// TwinCAT 3 PLC project tcext
// Title: TcExt
// Company: TcExt
// ProjectVersion: 0.2.3
// ProgramVersion: 3.1.4022.7
// libraries:
//   Tc2_Standard, * (Beckhoff Automation GmbH)
//   Tc2_System, * (Beckhoff Automation GmbH)
//   Tc2_Utilities, * (Beckhoff Automation GmbH)
//   Tc3_Module, * (Beckhoff Automation GmbH)
//   TcUnit, * (www.tcunit.org)
// project tree:
//   Files/ FileMemory.TcPOU, FileMemoryAction.TcDUT
//   Object/ BitAdrState.TcPOU, ModabsInt.TcPOU, Object.TcPOU
//   Tests/Files/ TestFileMemory.TcPOU
//   Tests/ MAIN.TcPOU, MAIN_TEST.TcPOU, PlcTask.TcTTO, TestBitAdrState.TcPOU, TestModabsInt.TcPOU
//   Tests/Timer/ TestSignalDutyCycleRecorder.TcPOU
//   Timer/ GetSystemTimeAsTime.TcPOU, SignalTimeRecorder.TcPOU, SignalDutyCycleRecorder.TcPOU, SimpleSignalTimeRecorder.TcPOU, SimpleTimeRecorder.TcPOU
//   Utils/ CompareReal.TcPOU, CrcCheck.TcPOU, FlashSignal.TcPOU, LockingRelay.TcPOU, TransitionController.TcPOU
//   Visu/ Colors.TcDUT, VisuElementProperties.TcDUT
// real-time tasks:
//   TASK PlcTask: cycle T#10ms, priority 20, ADS port 351

CONFIGURATION tcext
    RESOURCE PLC ON TwinCAT3
        TASK PlcTask(INTERVAL := T#10ms, PRIORITY := 20);
        PROGRAM MAIN WITH PlcTask : MAIN;
    END_RESOURCE
END_CONFIGURATION

// ---- Files/FileMemoryAction.TcDUT
{attribute 'qualified_only'}
{attribute 'strict'}
TYPE FileMemoryAction :
(
	UNLOCKED := 0,
  READ,
  WRITE
);
END_TYPE

// ---- Visu/Colors.TcDUT
{attribute 'qualified_only'}
{attribute 'strict'}
TYPE Colors :
(
  WHITE := 16#FFFFFF,
	BLACK := 16#000000,
	GRAY := 16#4C4C4C,
	LIGHT_GRAY := 16#C0C0C0,
	DARK_GRAY := 16#2D2D2D,
	RED := 16#FF0000,
	GREEN := 16#00FF00,
	YELLOW := 16#FFFF00,
  BLUE := 16#00BFFF
) DWORD := WHITE;
END_TYPE

// ---- Visu/VisuElementProperties.TcDUT
TYPE VisuElementProperties :
STRUCT
  color: DWORD;
  invisible: BOOL;
  int_value: INT;
END_STRUCT
END_TYPE

// ---- Tests/MAIN.TcPOU
{attribute 'hide'}
PROGRAM MAIN
VAR
END_VAR

{IF defined(TEST)}
MAIN_TEST();
{END_IF}

END_PROGRAM

// ---- Tests/MAIN_TEST.TcPOU
{attribute 'hide'}
PROGRAM MAIN_TEST
VAR
  test_file_memory: TestFileMemory;
  test_durchflusssensor: TestSignalDutyCycleRecorder;
  time_test: TIME;
  test_bit_adr_state: TestBitAdrState;
  test_modabs_int: TestModabsInt;
END_VAR

TcUnit.RUN();
time_test := TO_TIME(F_GetSystemTime()/10000);

END_PROGRAM

// ---- Tests/Files/TestFileMemory.TcPOU
{attribute 'call_after_init'}
FUNCTION_BLOCK TestFileMemory EXTENDS TcUnit.FB_TestSuite
VAR
END_VAR

//createFile();
set_path();
write_file();
read_non_existent_file();
read_existent_file();
write_and_read_simultaneously();
read_twice();
write_twice();
auto_write();
auto_write_time();

METHOD auto_write
VAR
  done: BOOL;
  error_id: UDINT;
END_VAR
VAR_INST
  file_memory: FileMemory;
  test_data: INT;
  test_data_first_read: INT;
  test_data_second_read: INT;
  counter: INT;
END_VAR
TEST('auto_write');

file_memory.path := 'c:\auto_write.be';
file_memory.auto_write(
  data_ptr:=ADR(test_data),
  data_size:=SIZEOF(test_data),
  done=>done,
  error_id=>error_id);

CASE counter OF
0:
  test_data := 135;
  counter := counter + 10;
10:
  IF done THEN
    counter := counter + 10;
  END_IF
20:
  file_memory.read(
    start:=TRUE,
    data_ptr:=ADR(test_data_first_read),
    data_size:=SIZEOF(test_data_first_read),
    done=>done,
    error_id=>error_id);
  IF done THEN
    counter := counter + 10;
  END_IF
30:
  file_memory.read(
    start:=FALSE,
    data_ptr:=0,
    data_size:=0);
  counter := counter + 10;
40:
  test_data := 246;
  counter := counter + 10;
50:
  IF done THEN
    counter := counter + 10;
  END_IF
60:
  file_memory.read(
    start:=TRUE,
    data_ptr:=ADR(test_data_second_read),
    data_size:=SIZEOF(test_data_second_read),
    done=>done,
    error_id=>error_id);
  IF done THEN
    AssertEquals_INT(135, test_data_first_read, 'Wrong values from auto_write file.');
    AssertEquals_INT(246, test_data_second_read, 'Wrong values from auto_write file.');
  
    TEST_FINISHED();
  END_IF
END_CASE
END_METHOD

METHOD auto_write_time
VAR
  done: BOOL;
  error_id: UDINT;
END_VAR
VAR_INST
  file_memory: FileMemory;
  test_data: INT;
  test_data_first_read: INT;
  test_data_second_read: INT;
  counter: INT;
  test_timer: TON;
END_VAR
TEST('auto_write_time');

file_memory.path := 'c:\auto_write_time.be';
file_memory.auto_write_time(
  data_ptr:=ADR(test_data),
  data_size:=SIZEOF(test_data),
  period:=T#2S,
  done=>done,
  error_id=>error_id);
test_timer(PT:=T#2.2S);

CASE counter OF
0:
  test_data := 135;
  counter := counter + 10;
10:
  test_timer(IN:=TRUE);
  IF test_timer.q THEN
    test_timer(IN:=FALSE);
    counter := counter + 10;
  END_IF
20:
  file_memory.read(
    start:=TRUE,
    data_ptr:=ADR(test_data_first_read),
    data_size:=SIZEOF(test_data_first_read),
    done=>done,
    error_id=>error_id);
  IF done THEN
    counter := counter + 10;
  END_IF
30:
  file_memory.read(
    start:=FALSE,
    data_ptr:=0,
    data_size:=0);
  counter := counter + 10;
40:
  test_data := 246;
  counter := counter + 10;
50:
  test_timer(IN:=TRUE);
  IF test_timer.q THEN
    test_timer(IN:=FALSE);
    counter := counter + 10;
  END_IF
60:
  file_memory.read(
    start:=TRUE,
    data_ptr:=ADR(test_data_second_read),
    data_size:=SIZEOF(test_data_second_read),
    done=>done,
    error_id=>error_id);
  IF done THEN
    AssertEquals_INT(135, test_data_first_read, 'Wrong values from auto_write file.');
    AssertEquals_INT(246, test_data_second_read, 'Wrong values from auto_write file.');
  
    TEST_FINISHED();
  END_IF
END_CASE
END_METHOD

METHOD PRIVATE createFile
VAR_INPUT
END_VAR
TEST('create_file');

TEST_FINISHED();
END_METHOD

METHOD read_existent_file
VAR
  done: BOOL;
  error_id: UDINT;
  
  expected: INT;
END_VAR
VAR_INST
  file_memory: FileMemory;
  test_data: INT;
END_VAR
TEST('read_existent_file');

IF IS_TEST_FINISHED('write_file') THEN
  file_memory.path := 'c:\test_file.be';
  
  file_memory.read(
    start:=TRUE,
    data_ptr:=ADR(test_data),
    data_size:=SIZEOF(test_data),
    done=>done,
    error_id=>error_id);
  
  IF done THEN
    expected := 37;
    AssertEquals_INT(expected, test_data, CONCAT('Wrong value. Check if file exists and contains 37. Error: ', TO_STRING(error_id)));
    
    TEST_FINISHED();
  END_IF
END_IF
END_METHOD

METHOD PRIVATE read_non_existent_file
VAR
  done: BOOL;
  error_id: UDINT;
  
  test_data: INT;
END_VAR
VAR_INST
    read_file: FileMemory;
END_VAR
TEST('read_non_existent_file');

read_file.path := 'c:\non_existent_file.be';

read_file.read(
  start:=TRUE,
  data_ptr:=ADR(test_data),
  data_size:=SIZEOF(test_data),
  done=>done,
  error_id=>error_id);

IF done THEN
  AssertTrue((error_id <> 0), 'No error although file non existent.');
  
  TEST_FINISHED();
END_IF
END_METHOD

METHOD read_twice
VAR
  done: BOOL;
  error_id: UDINT;
END_VAR
VAR_INST
  file_memory: FileMemory;
  test_data_first_read: INT;
  test_data_second_read: INT;
  counter: INT;
END_VAR
TEST('read_twice');

IF IS_TEST_FINISHED('write_file') AND IS_TEST_FINISHED('read_existent_file') THEN
  file_memory.path := 'c:\test_file.be';
  
  CASE counter OF
  0:
    file_memory.read(
      start:=TRUE,
      data_ptr:=ADR(test_data_first_read),
      data_size:=SIZEOF(test_data_first_read),
      done=>done,
      error_id=>error_id);
    IF done THEN
      counter := 10;
		END_IF
  10:
    file_memory.read(
      start:=FALSE,
      data_ptr:=0,
      data_size:=0);
    counter := 20;
  20:
    file_memory.read(
      start:=TRUE,
      data_ptr:=ADR(test_data_second_read),
      data_size:=SIZEOF(test_data_second_read),
      done=>done,
      error_id=>error_id);
    IF done THEN
      AssertEquals_INT(test_data_first_read, test_data_second_read, 'Wrong values from same file.');
    
      TEST_FINISHED();
		END_IF
	END_CASE
END_IF
END_METHOD

METHOD set_path
VAR
  actual: STRING;
  expected: STRING;
  
  file_memory: FileMemory;
END_VAR
TEST('set_path');

expected := 'c:\test.be';
file_memory.path := expected;
actual := file_memory.path;

AssertEquals_STRING(expected, actual, 'Path is broken.');

TEST_FINISHED();
END_METHOD

METHOD write_and_read_simultaneously
VAR
  done_write: BOOL;
  error_id_write: UDINT;
  done_read: BOOL;
  error_id_read: UDINT;
END_VAR
VAR_INST
  file_memory: FileMemory;
  test_data_write: INT;
  test_data_read: INT;
END_VAR
TEST('write_and_read_simultaneously');

file_memory.path := 'c:\test_file_2.be';

test_data_write := 123;
file_memory.write(
  start:=TRUE , 
  data_ptr:=ADR(test_data_write), 
  data_size:=SIZEOF(test_data_write), 
  done=>done_write, 
  error_id=>error_id_write);
file_memory.read(
  start:=TRUE , 
  data_ptr:=ADR(test_data_read), 
  data_size:=SIZEOF(test_data_read), 
  done=>done_read, 
  error_id=>error_id_read);
  
IF done_write AND done_read THEN
  AssertTrue((error_id_write = 0), CONCAT('Fehler beim simultanen Schreiben. Error: ', TO_STRING(error_id_write)));
  AssertTrue((error_id_read = 0), CONCAT('Fehler beim simultanen Lesen. Error: ', TO_STRING(error_id_read)));
  AssertEquals_INT(test_data_write, test_data_read, 'Geschriebene und gelesenen Daten ungleich.');
  
  TEST_FINISHED();
END_IF
END_METHOD

METHOD write_file
VAR
  done: BOOL;
  error_id: UDINT;
END_VAR
VAR_INST
  file_memory: FileMemory;
  test_data: INT;
END_VAR
TEST('write_file');

file_memory.path := 'c:\test_file.be';

test_data := 37;

file_memory.write(
  start:=TRUE,
  data_ptr:=ADR(test_data),
  data_size:=SIZEOF(test_data),
  done=>done,
  error_id=>error_id);
  
IF done THEN
  AssertEquals_UDINT(0, error_id, CONCAT('File could not be written. Error: ', TO_STRING(error_id)));
  
  TEST_FINISHED();
END_IF
END_METHOD

METHOD write_twice
VAR
  done: BOOL;
  error_id: UDINT;
END_VAR
VAR_INST
  file_memory: FileMemory;
  test_data_first_write: INT;
  test_data_second_write: INT;
  test_data_first_read: INT;
  test_data_second_read: INT;
  counter: INT;
END_VAR
TEST('write_twice');

file_memory.path := 'c:\write_twice.be';

test_data_first_write := 123;
test_data_second_write := 456;
CASE counter OF
0:
  file_memory.write(
    start:=TRUE,
    data_ptr:=ADR(test_data_first_write),
    data_size:=SIZEOF(test_data_first_write),
    done=>done,
    error_id=>error_id);
  IF done THEN
    counter := 10;
  END_IF
10:
  file_memory.write(
    start:=FALSE,
    data_ptr:=0,
    data_size:=0);
  counter := 20;
20:
  file_memory.read(
    start:=TRUE,
    data_ptr:=ADR(test_data_first_read),
    data_size:=SIZEOF(test_data_first_read),
    done=>done,
    error_id=>error_id);
  IF done THEN
    counter := 30;
  END_IF
30:
  file_memory.read(
    start:=FALSE,
    data_ptr:=0,
    data_size:=0);
  counter := 40;
40:
  file_memory.write(
    start:=TRUE,
    data_ptr:=ADR(test_data_second_write),
    data_size:=SIZEOF(test_data_second_write),
    done=>done,
    error_id=>error_id);
  IF done THEN
    counter := 50;
  END_IF
50:
  file_memory.write(
    start:=FALSE,
    data_ptr:=0,
    data_size:=0);
  counter := 60;
60:
  file_memory.read(
    start:=TRUE,
    data_ptr:=ADR(test_data_second_read),
    data_size:=SIZEOF(test_data_second_read),
    done=>done,
    error_id=>error_id);
  IF done THEN
    AssertEquals_INT(test_data_first_write, test_data_first_read, 'Wrong values from same file.');
    AssertEquals_INT(test_data_second_write, test_data_second_read, 'Wrong values from same file.');
  
    TEST_FINISHED();
  END_IF
END_CASE
END_METHOD

END_FUNCTION_BLOCK

// ---- Files/FileMemory.TcPOU
FUNCTION_BLOCK FileMemory EXTENDS Object
VAR
  file_path: Tc2_System.T_MaxString;
  
  fb_file_open: Tc2_System.FB_FileOpen;
  fb_file_close: Tc2_System.FB_FileClose;
  fb_file_read: Tc2_System.FB_FileRead;
  fb_file_write: Tc2_System.FB_FileWrite;
  
  t_timeout_read: TIME := T#2S;
  t_timeout_write: TIME := T#2S;
  
  lock_action: FileMemoryAction;
  
  write_period_timer: Tc2_Standard.TP;
  crc_check: CrcCheck;
  _mode_read: DWORD := Tc2_System.FOPEN_MODEREAD OR Tc2_System.FOPEN_MODEBINARY;
  _mode_write: DWORD := Tc2_System.FOPEN_MODEWRITE OR Tc2_System.FOPEN_MODEBINARY;
END_VAR

METHOD auto_write
VAR_INPUT
  data_ptr: POINTER TO BYTE;
  data_size: UDINT;
END_VAR
VAR_OUTPUT
  done: BOOL;
  error_id: UDINT;
END_VAR
VAR
  crc_changed: BOOL;
END_VAR
VAR_INST
  act_crc: UINT;
  previous_crc: UINT;
END_VAR
write(
  start:=crc_check.data_changed(data_ptr, data_size), 
  data_ptr:=data_ptr, 
  data_size:=data_size,
  done=>done,
  error_id=>error_id);
  
IF done THEN
  crc_check.reset();
END_IF
END_METHOD

METHOD auto_write_time
VAR_INPUT
  data_ptr: POINTER TO BYTE;
  data_size: UDINT;
  period: TIME;
END_VAR
VAR_OUTPUT
  done: BOOL;
  error_id: UDINT;
END_VAR
write_period_timer(IN:=NOT write_period_timer.Q, PT:=period);

write(
  start:=NOT write_period_timer.q AND crc_check.data_changed(data_ptr, data_size), 
  data_ptr:=data_ptr, 
  data_size:=data_size,
  done=>done,
  error_id=>error_id);
  
IF NOT write_period_timer.q THEN
  crc_check.reset();
END_IF
END_METHOD

PROPERTY PUBLIC busy_reading : BOOL
GET
busy_reading := THIS^.lock_action = FileMemoryAction.READ;
END_GET
END_PROPERTY

PROPERTY PUBLIC busy_writing : BOOL
GET
busy_writing := THIS^.lock_action = FileMemoryAction.WRITE;
END_GET
END_PROPERTY

METHOD file_close
VAR_INPUT
  start: BOOL;
  file_handler: UINT;
END_VAR
VAR_OUTPUT
  done: BOOL;
  error_id: UDINT;
END_VAR
fb_file_close(
  bExecute:=start,
  hFile:=file_handler);

IF NOT fb_file_close.bBusy THEN
  done := TRUE;
  IF fb_file_close.bError THEN
    error_id := fb_file_close.nErrId;
  END_IF
END_IF
END_METHOD

METHOD PRIVATE file_open: UINT
VAR_INPUT
  start: BOOL;
  mode: DWORD;
END_VAR
VAR_OUTPUT
  done: BOOL;
  error_id: UDINT;
END_VAR
fb_file_open(
  bExecute:=start,
  sPathName:=path,
  nMode:=mode);

file_open := 0;
IF NOT fb_file_open.bBusy THEN
  done := TRUE;
  IF fb_file_open.bError THEN
    error_id := fb_file_open.nErrId;
  ELSE
    file_open := fb_file_open.hFile;
  END_IF
END_IF
END_METHOD

METHOD PRIVATE file_read
VAR_INPUT
  start: BOOL;
  file_handler: UINT;
  data_ptr: POINTER TO BYTE;
  data_size: UDINT;
END_VAR
VAR_OUTPUT
  done: BOOL;
  error_id: UDINT;
END_VAR
fb_file_read(
  bExecute:=start,
  hFile:=file_handler,
  pReadBuff:=data_ptr,
  cbReadLen:=data_size);

IF NOT fb_file_read.bBusy THEN
  done := TRUE;
  IF fb_file_read.bError THEN
    error_id := fb_file_read.nErrId;
  END_IF
END_IF
END_METHOD

METHOD PRIVATE file_write
VAR_INPUT
  start: BOOL;
  file_handler: UINT;
  data_ptr: POINTER TO BYTE;
  data_size: UDINT;
END_VAR
VAR_OUTPUT
  done: BOOL;
  error_id: UDINT;
END_VAR
fb_file_write(
  bExecute:=start,
  hFile:=file_handler,
  pWriteBuff:=data_ptr,
  cbWriteLen:=data_size);

IF NOT fb_file_write.bBusy THEN
  done := TRUE;
  IF fb_file_write.bError THEN
    error_id := fb_file_write.nErrId;
  END_IF
END_IF
END_METHOD

METHOD PRIVATE lock
VAR_INPUT
  lock_action: FileMemoryAction;
END_VAR
THIS^.lock_action := lock_action;
END_METHOD

METHOD PRIVATE locked : BOOL
VAR_INPUT
  lock_action: FileMemoryAction;
END_VAR
locked := (THIS^.lock_action <> FileMemoryAction.UNLOCKED) AND (THIS^.lock_action <> lock_action);
END_METHOD

PROPERTY PUBLIC mode_read : DWORD
GET
mode_read := _mode_read;
END_GET
SET
_mode_read := mode_read;
END_SET
END_PROPERTY

PROPERTY PUBLIC mode_write : DWORD
GET
mode_write := _mode_write;
END_GET
SET
_mode_write := mode_write;
END_SET
END_PROPERTY

PROPERTY path : T_MaxString
GET
path := file_path;
END_GET
SET
file_path := path;
END_SET
END_PROPERTY

METHOD read
VAR_INPUT
  start: BOOL;
  data_ptr: POINTER TO BYTE;
  data_size: UDINT;
END_VAR
VAR_OUTPUT
  done: BOOL;
  error_id: UDINT;
  file_not_found: BOOL;
END_VAR
VAR
  next_state: BOOL;
  done_temp: BOOL;
END_VAR
VAR_INST
  file_handler: UINT;
  lr_start: LockingRelay;
  done_mem: BOOL;
  error_id_mem: UDINT;
  timeout_timer: Tc2_Standard.TON;
  timeout_start: BOOL;
  
  open_transition: TransitionController;
  read_transition: TransitionController;
  close_transition: TransitionController;
  
  finished: BOOL;
  
  counter: INT;
END_VAR
lr_start.clk := start;
timeout_timer(IN:=timeout_start, PT:=timeout_read);
IF timeout_timer.Q THEN
  counter := -1;
  error_id_mem := 16#010000;
END_IF

CASE counter OF
0:
  done_mem := TRUE;
  IF lr_start.q THEN
    lr_start.reset := TRUE;
    done_mem := FALSE;
    error_id_mem := 0;
    counter := counter + 10;
  END_IF
10:
  IF NOT locked(FileMemoryAction.READ) THEN
    timeout_start := FALSE;
    reset_file_fbs();
    lock(FileMemoryAction.READ);
    counter := counter + 10;
  END_IF
20:
  file_handler := file_open(start:=TRUE, mode:=mode_read, done=>next_state, error_id=>error_id_mem);
30:
  file_open(start:=FALSE, mode:=0, done=>next_state);
40:
  file_read(start:=TRUE, file_handler:=file_handler, data_ptr:=data_ptr, data_size:=data_size, 
    done=>next_state, error_id=>error_id_mem);
50:
  file_read(start:=FALSE, file_handler:=0, data_ptr:=0, data_size:=0, done=>next_state);
60:
  file_close(start:=TRUE, file_handler:=file_handler, done=>next_state, error_id=>error_id_mem);
70:
  file_close(start:=FALSE, file_handler:=0, done=>next_state);
ELSE
  timeout_start := FALSE;
  counter := 0;
  unlock();
END_CASE
IF next_state AND (error_id_mem <> 0) THEN
  counter := -1;
ELSIF next_state THEN
  counter := counter + 10;
END_IF

done := done_mem;
error_id := error_id_mem;
file_not_found := error_id = 16#070C;
END_METHOD

METHOD PRIVATE reset_file_fbs
file_open(
  start:=FALSE,
  mode:=0);
file_write(
  start:=FALSE,
  file_handler:=0,
  data_ptr:=0,
  data_size:=0);
file_read(
    start:=FALSE,
    file_handler:=0,
    data_ptr:=0,
    data_size:=0);
// it looks like fb_file_close needs to be called at least once after successfully
// closing a file before starting it again (at least with version 4022.25)
file_close(
  start:=FALSE,
  file_handler:=0);
END_METHOD

PROPERTY timeout_read : TIME
GET
timeout_read := t_timeout_read;
END_GET
SET
t_timeout_read := timeout_read;
END_SET
END_PROPERTY

PROPERTY timeout_write : TIME
GET
timeout_write := t_timeout_write;
END_GET
SET
t_timeout_write := timeout_write;
END_SET
END_PROPERTY

METHOD PRIVATE unlock
lock(FileMemoryAction.UNLOCKED);
END_METHOD

METHOD write
VAR_INPUT
  start: BOOL;
  data_ptr: POINTER TO BYTE;
  data_size: UDINT;
END_VAR
VAR_OUTPUT
  done: BOOL;
  error_id: UDINT;
END_VAR
VAR
  next_state: BOOL;
END_VAR
VAR_INST
  file_handler: UINT;
  lr_start: LockingRelay;
  done_mem: BOOL;
  error_id_mem: UDINT;
  counter: INT;
  timeout_timer: Tc2_Standard.TON;
  timeout_start: BOOL;
END_VAR
lr_start.clk := start;
timeout_timer(IN:=timeout_start, PT:=timeout_write);
IF timeout_timer.Q THEN
  counter := -1;
  error_id_mem := 16#010000;
END_IF

CASE counter OF
0:
  done_mem := TRUE;
  IF lr_start.q THEN
    lr_start.reset := TRUE;
    done_mem := FALSE;
    error_id_mem := 0;
    counter := counter + 10;
  END_IF
10:
  IF NOT locked(FileMemoryAction.WRITE) THEN
    timeout_start := FALSE;
    reset_file_fbs();
    lock(FileMemoryAction.WRITE);
    counter := counter + 10;
  END_IF
20:
  file_handler := file_open(start:=TRUE, mode:=mode_write, done=>next_state, error_id=>error_id_mem);
30:
  file_open(start:=FALSE, mode:=0, done=>next_state);
40:
  file_write(start:=TRUE, file_handler:=file_handler, data_ptr:=data_ptr, data_size:=data_size, 
    done=>next_state, error_id=>error_id_mem);
50:
  file_write(start:=FALSE, file_handler:=0, data_ptr:=0, data_size:=0, done=>next_state);
60:
  file_close(start:=TRUE, file_handler:=file_handler, done=>next_state, error_id=>error_id_mem);
70:
  file_close(start:=FALSE, file_handler:=0, done=>next_state);
ELSE
  timeout_start := FALSE;
  counter := 0;
  unlock();
END_CASE
IF next_state AND (error_id_mem <> 0) THEN
  counter := -1;
ELSIF next_state THEN
  counter := counter + 10;
END_IF

done := done_mem;
error_id := error_id_mem;
END_METHOD

END_FUNCTION_BLOCK

// ---- Object/Object.TcPOU
{attribute 'reflection'}
FUNCTION_BLOCK Object
VAR_OUTPUT 
  busy: BOOL;
	done: BOOL;
  ready: BOOL;
//	error: BOOL;
  error_id: UDINT;
END_VAR
VAR
  {attribute 'instance-path'}
  {attribute 'noinit'}
  fb_id: STRING(255);
END_VAR

END_FUNCTION_BLOCK

// ---- Utils/CrcCheck.TcPOU
FUNCTION_BLOCK CrcCheck
VAR_INPUT
END_VAR
VAR_OUTPUT
END_VAR
VAR
  act_crc: UINT;
  previous_crc: UINT;
END_VAR

METHOD data_changed : BOOL
VAR_INPUT
  data_ptr: POINTER TO BYTE;
  data_size: UDINT;
END_VAR
act_crc := F_DATA_TO_CRC16_CCITT(data_ptr, data_size, 0);
data_changed := act_crc <> previous_crc;
END_METHOD

METHOD reset
VAR_INPUT
END_VAR
previous_crc := act_crc;
END_METHOD

END_FUNCTION_BLOCK

// ---- Utils/LockingRelay.TcPOU
FUNCTION_BLOCK LockingRelay EXTENDS Object
VAR_INPUT
END_VAR
VAR_OUTPUT
END_VAR
VAR
  _clk: BOOL;
  r_clk: R_TRIG;
END_VAR

PROPERTY clk : BOOL
SET
r_clk(CLK:=clk);
IF r_clk.Q THEN
  _clk := TRUE;
ELSIF NOT clk THEN
  _clk := FALSE;
END_IF
END_SET
END_PROPERTY

PROPERTY q : BOOL
GET
q := _clk;
END_GET
END_PROPERTY

PROPERTY reset : BOOL
SET
IF reset THEN
  _clk := FALSE;
END_IF
END_SET
END_PROPERTY

END_FUNCTION_BLOCK

// ---- Utils/TransitionController.TcPOU
FUNCTION_BLOCK TransitionController
VAR_INPUT
  done: BOOL;
  error: BOOL;
  error_id: UDINT;
END_VAR
VAR_OUTPUT
  execute_level: BOOL;
  execute_trigger: BOOL;
END_VAR
VAR
  lr_execute: LockingRelay;
  r_execute: R_TRIG;
  _execute: BOOL;
  lr_done: LockingRelay;
  lr_error: LockingRelay;
END_VAR

METHOD fire
VAR_INPUT
  execute: BOOL;
END_VAR
lr_execute.clk := execute;
r_execute(CLK:=execute);
IF r_execute.Q THEN
  _execute := TRUE;
END_IF

execute_trigger := r_execute.q;

execute_level := lr_execute.q;
END_METHOD

PROPERTY transition : BOOL
GET
IF _execute THEN
  lr_done.clk := done;
END_IF
lr_error.clk := (error_id <> 0) OR error;
transition := lr_done.q AND NOT lr_error.q;
IF transition THEN
  lr_done.reset := TRUE;
  lr_error.reset := TRUE;
  _execute := FALSE;
END_IF
END_GET
END_PROPERTY

END_FUNCTION_BLOCK

// ---- Tests/Timer/TestSignalDutyCycleRecorder.TcPOU
FUNCTION_BLOCK TestSignalDutyCycleRecorder EXTENDS TcUnit.FB_TestSuite
VAR_INPUT
END_VAR
VAR_OUTPUT
END_VAR
VAR
END_VAR

GibtNichtsAusWennNeuErstellt();
DurchflussIOWenn100ProzentAnImSelbenZyklus();
DurchflussNIOWenn100ProzentAusImSelbenZyklus();
DurchflussNIOWenn60zu40ProzentAusInMehrerenZyklen();
DurchflussIOWenn60zu40ProzentAnInMehrerenZyklen();
DurchflussAufnahmeMehrmalsDurchfuehren();
AufnahmeNachTimeoutAbbrechen();
AufnahmeNachTimeoutAbbrechenUndStoppenIstTrotzdemNIO();
AufnahmeNachResetEinerFehlerhaftenAufnahme();
AufnahmeBeruecksichtigtStartverzoegerung();
// negativer Tastgrad
// positiver Tastgrad

METHOD AufnahmeBeruecksichtigtStartverzoegerung
VAR_INPUT
END_VAR
VAR_INST
  sensor: SignalDutyCycleRecorder;
  aufnahmedauer: TIME;
  t_aufnahmedauer: TON;
  zaehler: INT;
END_VAR
TEST('AufnahmeBeruecksichtigtStartverzoegerung');

aufnahmedauer := T#1S;
t_aufnahmedauer(IN:=TRUE, PT:=aufnahmedauer);

sensor.record_delay := T#500MS;
sensor.signal := t_aufnahmedauer.ET <= T#700MS;
sensor.set_duty_cycle_in_percent := 50.0;

sensor.record(execute:=NOT t_aufnahmedauer.Q);

IF t_aufnahmedauer.Q THEN
  AssertTrue(sensor.recording_finished, 'Normaler Ablauf');
  AssertFalse(sensor.duty_cycle_ok, 'Aufgrund der Startverzoegerung darf der Durchfluss nicht i.O. sein');
  AssertFalse(sensor.error, 'Kein Fehler');
  
  TEST_FINISHED();
END_IF
END_METHOD

METHOD AufnahmeNachResetEinerFehlerhaftenAufnahme
VAR_INPUT
END_VAR
VAR_INST
  sensor: SignalDutyCycleRecorder;
  timeoutdauer: TIME;
  zaehler: INT;
END_VAR
TEST('AufnahmeNachResetEinerFehlerhaftenAufnahme');

timeoutdauer := T#1S;

sensor.record_delay := T#0S;
sensor.signal := TRUE;
sensor.timeout := timeoutdauer;

CASE zaehler OF
0:
  sensor.record(execute:=TRUE);
  
  IF sensor.error THEN
    sensor.record(execute:=FALSE);
  
    AssertTrue(sensor.recording_finished, 'Timeout-Fehler, daher ist die Aufnahme beendet');
    AssertFalse(sensor.duty_cycle_ok, 'Bei Fehler darf der Durchfluss nicht i.O. sein');
    AssertTrue(sensor.error, 'Timeout-Fehler eingetreten');
    
    zaehler := zaehler + 1;
  END_IF
1:
  sensor.reset();
  AssertFalse(sensor.error, 'Fehler wurde resettet');
  
  zaehler := zaehler + 1;
2:
  sensor.record(execute:=TRUE);
  
  AssertFalse(sensor.recording_finished, 'Timeout-Fehler, daher darf die Aufnahme auch nach einem stopp nicht starten');
  AssertFalse(sensor.duty_cycle_ok, 'Bei Fehler darf der Durchfluss nicht i.O. sein');
  AssertFalse(sensor.error, 'Timeout-Fehler eingetreten');
  
  zaehler := zaehler + 1;
3:
  sensor.record(execute:=FALSE);
  
  AssertTrue(sensor.recording_finished, 'Wurde korrekt gestoppt');
  AssertTrue(sensor.duty_cycle_ok, 'Sollte i.O. sein');
  AssertFalse(sensor.error, 'Timeout-Fehler eingetreten');
  
  TEST_FINISHED();
END_CASE
END_METHOD

METHOD AufnahmeNachTimeoutAbbrechen
VAR_INPUT
END_VAR
VAR_INST
  sensor: SignalDutyCycleRecorder;
  timeoutdauer: TIME;
  t_timeout_vor: TON;
  t_timeout_nach: TON;
  zaehler: INT;
END_VAR
TEST('AufnahmeNachTimeoutAbbrechen');

timeoutdauer := T#1S;
t_timeout_vor(IN:=TRUE, PT:=timeoutdauer-T#100MS);
t_timeout_nach(IN:=TRUE, PT:=timeoutdauer+T#100MS);

sensor.record_delay := T#0S;
sensor.timeout := timeoutdauer;

sensor.record(execute:=TRUE);

CASE zaehler OF
0:  
  IF t_timeout_vor.Q THEN
    AssertFalse(sensor.recording_finished, 'Aufnahme laeuft');
    AssertFalse(sensor.duty_cycle_ok, 'Aufnahme laeuft, daher muss es aus sein');
    AssertFalse(sensor.error, 'Es darf kein Fehler anliegen');
    
    zaehler := zaehler + 1;
  END_IF
1:
  IF t_timeout_nach.Q THEN
    AssertTrue(sensor.recording_finished, 'Timeout-Fehler, daher ist die Aufnahme beendet');
    AssertFalse(sensor.duty_cycle_ok, 'Bei Fehler darf der Durchfluss nicht i.O. sein');
    AssertTrue(sensor.error, 'Timeout-Fehler eingetreten');
    
    TEST_FINISHED();
  END_IF
END_CASE
END_METHOD

METHOD AufnahmeNachTimeoutAbbrechenUndStoppenIstTrotzdemNIO
VAR_INPUT
END_VAR
VAR_INST
  sensor: SignalDutyCycleRecorder;
  timeoutdauer: TIME;
  zaehler: INT;
END_VAR
TEST('AufnahmeNachTimeoutAbbrechenUndStoppenIstTrotzdemNIO');

timeoutdauer := T#1S;

sensor.record_delay := T#0S;
sensor.signal := TRUE;
sensor.timeout := timeoutdauer;

CASE zaehler OF
0:
  sensor.record(execute:=TRUE);
  
  IF sensor.error THEN
    sensor.record(execute:=FALSE);
  
    AssertTrue(sensor.recording_finished, 'Timeout-Fehler, daher ist die Aufnahme beendet');
    AssertFalse(sensor.duty_cycle_ok, 'Bei Fehler darf der Durchfluss nicht i.O. sein');
    AssertTrue(sensor.error, 'Timeout-Fehler eingetreten');
    
    zaehler := zaehler + 1;
  END_IF
1:
  sensor.record(execute:=TRUE);
  
  AssertTrue(sensor.recording_finished, 'Timeout-Fehler, daher darf die Aufnahme auch nach einem stopp nicht starten');
  AssertFalse(sensor.duty_cycle_ok, 'Bei Fehler darf der Durchfluss nicht i.O. sein');
  AssertTrue(sensor.error, 'Timeout-Fehler eingetreten');
  
  TEST_FINISHED();
END_CASE
END_METHOD

METHOD DurchflussAufnahmeMehrmalsDurchfuehren
VAR_INPUT
END_VAR
VAR_INST
  sensor: SignalDutyCycleRecorder;
  aufnahmedauer: TIME;
  t_aufnahmedauer: TON;
  zaehler: INT;
END_VAR
TEST('DurchflussAufnahmeMehrmalsDurchfuehren');

aufnahmedauer := T#500MS;

CASE zaehler OF
0:
  t_aufnahmedauer(IN:=TRUE, PT:=aufnahmedauer);

  sensor.record_delay := T#0S;
  sensor.signal := t_aufnahmedauer.ET <= T#200MS;
  sensor.set_duty_cycle_in_percent := 50.0;
  
  sensor.record(execute:=NOT t_aufnahmedauer.Q);
  
  IF NOT t_aufnahmedauer.Q THEN
    AssertFalse(sensor.recording_finished, 'Aufnahme laeuft');
  ELSE
    AssertTrue(sensor.recording_finished, '1. Aufnahme gestartet und sofort beendet');
    AssertFalse(sensor.duty_cycle_ok, '1. Durchfluss muss n.i.O. sein');
    AssertFalse(sensor.error, '1. Es darf kein Fehler anliegen');
    
    t_aufnahmedauer(IN:=FALSE);
    zaehler := zaehler + 1;
  END_IF
1:
  t_aufnahmedauer(IN:=TRUE, PT:=aufnahmedauer);

  sensor.record_delay := T#0S;
  sensor.signal := t_aufnahmedauer.ET >= T#80MS;
  sensor.set_duty_cycle_in_percent := 80.0;
  
  sensor.record(execute:=NOT t_aufnahmedauer.Q);
  
  IF NOT t_aufnahmedauer.Q THEN
    AssertFalse(sensor.recording_finished, 'Aufnahme laeuft');
    AssertFalse(sensor.duty_cycle_ok, 'Aufnahme laeuft, daher muss es aus sein');
    AssertFalse(sensor.error, 'Es darf kein Fehler anliegen');
  ELSE
    AssertTrue(sensor.recording_finished, '2. Aufnahme gestartet und sofort beendet');
    AssertTrue(sensor.duty_cycle_ok, '2. Durchfluss muss i.O. sein');
    AssertFalse(sensor.error, '2. Es darf kein Fehler anliegen');
    
    TEST_FINISHED();
  END_IF
END_CASE
END_METHOD

METHOD DurchflussIOWenn100ProzentAnImSelbenZyklus
VAR_INPUT
END_VAR
VAR_INST
  sensor: SignalDutyCycleRecorder;
END_VAR
TEST('DurchflussIOWenn100ProzentAnImSelbenZyklus');

sensor.record_delay := T#0S;
sensor.signal := TRUE;
sensor.set_duty_cycle_in_percent := 100.0;

sensor.record(execute:=TRUE);

sensor.record(execute:=FALSE);

AssertTrue(sensor.recording_finished, 'Aufnahme gestartet und sofort beendet');
AssertTrue(sensor.duty_cycle_ok, 'Durchfluss muss i.O. sein');
AssertFalse(sensor.error, 'Es darf kein Fehler anliegen');

TEST_FINISHED();
END_METHOD

METHOD DurchflussIOWenn60zu40ProzentAnInMehrerenZyklen
VAR_INPUT
END_VAR
VAR_INST
  sensor: SignalDutyCycleRecorder;
  aufnahmedauer: TIME;
  t_aufnahmedauer: TON;
END_VAR
TEST('DurchflussIOWenn60zu40ProzentAnInMehrerenZyklen');

aufnahmedauer := T#1S;
t_aufnahmedauer(IN:=TRUE, PT:=aufnahmedauer);

sensor.record_delay := T#0S;
sensor.signal := t_aufnahmedauer.ET <= T#600MS;
sensor.set_duty_cycle_in_percent := 50.0;

sensor.record(execute:=NOT t_aufnahmedauer.Q);

IF NOT t_aufnahmedauer.Q THEN
  AssertFalse(sensor.recording_finished, 'Aufnahme laeuft');
ELSE
  AssertTrue(sensor.recording_finished, 'Aufnahme gestartet und sofort beendet');
  AssertTrue(sensor.duty_cycle_ok, 'Durchfluss muss i.O. sein');
  AssertFalse(sensor.error, 'Es darf kein Fehler anliegen');
  
  TEST_FINISHED();
END_IF
END_METHOD

METHOD DurchflussNIOWenn100ProzentAusImSelbenZyklus
VAR_INPUT
END_VAR
VAR_INST
  sensor: SignalDutyCycleRecorder;
END_VAR
TEST('DurchflussNIOWenn100ProzentAusImSelbenZyklus');

sensor.record_delay := T#0S;
sensor.signal := FALSE;
sensor.set_duty_cycle_in_percent := 100.0;

sensor.record(execute:=TRUE);

sensor.record(execute:=FALSE);

AssertTrue(sensor.recording_finished, 'Aufnahme gestartet und sofort beendet');
AssertFalse(sensor.duty_cycle_ok, 'Durchfluss muss n.i.O. sein');
AssertFalse(sensor.error, 'Es darf kein Fehler anliegen');

TEST_FINISHED();
END_METHOD

METHOD DurchflussNIOWenn60zu40ProzentAusInMehrerenZyklen
VAR_INPUT
END_VAR
VAR_INST
  sensor: SignalDutyCycleRecorder;
  aufnahmedauer: TIME;
  t_aufnahmedauer: TON;
END_VAR
TEST('DurchflussNIOWenn60zu40ProzentAusInMehrerenZyklen');

aufnahmedauer := T#1S;
t_aufnahmedauer(IN:=TRUE, PT:=aufnahmedauer);

sensor.record_delay := T#0S;
sensor.signal := t_aufnahmedauer.ET >= T#600MS;
sensor.set_duty_cycle_in_percent := 50.0;

sensor.record(execute:=NOT t_aufnahmedauer.Q);

IF NOT t_aufnahmedauer.Q THEN
  AssertFalse(sensor.recording_finished, 'Aufnahme laeuft');
ELSE
  AssertTrue(sensor.recording_finished, 'Aufnahme gestartet und sofort beendet');
  AssertFalse(sensor.duty_cycle_ok, 'Durchfluss muss n.i.O. sein');
  AssertFalse(sensor.error, 'Es darf kein Fehler anliegen');
  
  TEST_FINISHED();
END_IF
END_METHOD

METHOD GibtNichtsAusWennNeuErstellt
VAR_INPUT
END_VAR
VAR_INST
  sensor: SignalDutyCycleRecorder;
END_VAR
TEST('GibtNichtsAusWennNeuErstellt');

sensor.record(execute:=FALSE);

sensor.record(execute:=FALSE);

AssertFalse(sensor.recording_finished, 'Keine Aufnahme gestartet, daher kann auch keine beendet sein');
AssertFalse(sensor.duty_cycle_ok, 'Nie gestartet');
AssertFalse(sensor.error, 'Es darf kein Fehler anliegen');

TEST_FINISHED();
END_METHOD

END_FUNCTION_BLOCK

// ---- Timer/SignalDutyCycleRecorder.TcPOU
(*
Der Soll-Tastgrad in Prozent gibt das Verhaeltnis der Sensorzustaende An zu Aus waehrend einer Aufnahme an.
*)
FUNCTION_BLOCK SignalDutyCycleRecorder
VAR_INPUT
  signal: BOOL;
END_VAR
VAR_OUTPUT
  recording_finished: BOOL;
  duty_cycle_ok: BOOL;
  error: BOOL;
END_VAR
VAR
  _record_delay: TIME := T#1S;
  _timeout: TIME := T#10S;
  _set_duty_cycle_in_percent: REAL := 90.0;
  signal_recorder: SignalTimeRecorder;
END_VAR

METHOD record
VAR_INPUT
  execute: BOOL;
END_VAR
VAR
  start_recording: BOOL;
END_VAR
VAR_INST
  t_timeout: TON;
  f_started_recording: F_TRIG;
  r_execute: R_TRIG;
END_VAR
r_execute(CLK:=execute);
IF r_execute.Q AND NOT error THEN
  recording_finished := FALSE;
  signal_recorder.record(execute:=FALSE);
  signal_recorder.reset();
END_IF

t_timeout(IN:=signal_recorder.started_recording, PT:=timeout);
IF t_timeout.Q THEN
  error := TRUE;
END_IF

start_recording := execute AND NOT error;

signal_recorder.record_delay := record_delay;
signal_recorder.signal := signal;
signal_recorder.record(execute:=start_recording);

f_started_recording(CLK:=signal_recorder.started_recording);
IF f_started_recording.Q THEN
  recording_finished := TRUE;
  duty_cycle_ok := signal_recorder.on_ratio * 100.0 >= set_duty_cycle_in_percent AND NOT error;
END_IF
END_METHOD

{attribute 'monitoring' := 'call'}
PROPERTY record_delay : TIME
GET
record_delay := _record_delay;
END_GET
SET
_record_delay := record_delay;
END_SET
END_PROPERTY

METHOD reset
VAR_INPUT
END_VAR
error := FALSE;
signal_recorder.reset();
END_METHOD

{attribute 'monitoring' := 'call'}
PROPERTY set_duty_cycle_in_percent : REAL
GET
set_duty_cycle_in_percent := _set_duty_cycle_in_percent;
END_GET
SET
VAR
  tastgrad: REAL;
END_VAR
IF set_duty_cycle_in_percent < 0 THEN
  tastgrad := 0.0;
ELSIF set_duty_cycle_in_percent > 100.0 THEN
  tastgrad := 100.0;
ELSE
  tastgrad := set_duty_cycle_in_percent;
END_IF
_set_duty_cycle_in_percent := tastgrad;
END_SET
END_PROPERTY

{attribute 'monitoring' := 'call'}
PROPERTY timeout : TIME
GET
timeout := _timeout;
END_GET
SET
_timeout := timeout;
END_SET
END_PROPERTY

END_FUNCTION_BLOCK

// ---- Timer/SignalTimeRecorder.TcPOU
FUNCTION_BLOCK SignalTimeRecorder
VAR_INPUT
END_VAR
VAR_OUTPUT
END_VAR
VAR
  _record_delay: TIME;
  _signal: BOOL;
  _signal_filtertime: TIME;
  filtertime: TIME;
  
  _duration_on_in_ms: ULINT;
  _timestamp_on_in_ms: ULINT;
  _duration_off_in_ms: ULINT;
  _timestamp_off_in_ms: ULINT;
  t_record_delay: TON;
  t_signal_filtertime: TON;
END_VAR

{attribute 'monitoring' := 'call'}
PROPERTY PUBLIC act_duration_off_in_ms : ULINT
GET
act_duration_off_in_ms := duration_off_in_ms;
IF timestamp_off_in_ms > 0 THEN
  act_duration_off_in_ms := act_duration_off_in_ms + (act_timestamp_in_ms - timestamp_off_in_ms);
END_IF
END_GET
END_PROPERTY

{attribute 'monitoring' := 'call'}
PROPERTY PUBLIC act_duration_on_in_ms : ULINT
GET
act_duration_on_in_ms := duration_on_in_ms;
IF timestamp_on_in_ms > 0 THEN
  act_duration_on_in_ms := act_duration_on_in_ms + (act_timestamp_in_ms - timestamp_on_in_ms);
END_IF
END_GET
END_PROPERTY

{attribute 'monitoring' := 'call'}
PROPERTY act_record_duration_in_ms : ULINT
GET
act_record_duration_in_ms := act_duration_on_in_ms + act_duration_off_in_ms;
END_GET
END_PROPERTY

{attribute 'monitoring' := 'call'}
PROPERTY PRIVATE act_timestamp_in_ms : ULINT
GET
act_timestamp_in_ms := F_GetSystemTime() / 10000;
END_GET
END_PROPERTY

METHOD PRIVATE apply_duration
VAR_INPUT
END_VAR
IF timestamp_on_in_ms > 0 THEN
  duration_on_in_ms := duration_on_in_ms + (act_timestamp_in_ms - timestamp_on_in_ms);
  timestamp_on_in_ms := 0;
END_IF
IF timestamp_off_in_ms > 0 THEN
  duration_off_in_ms := duration_off_in_ms + (act_timestamp_in_ms - timestamp_off_in_ms);
  timestamp_off_in_ms := 0;
END_IF
END_METHOD

{attribute 'monitoring' := 'call'}
PROPERTY duration_off : TIME
GET
duration_off := TO_TIME(act_duration_off_in_ms);
END_GET
END_PROPERTY

{attribute 'monitoring' := 'call'}
PROPERTY PUBLIC duration_off_in_ms : ULINT
GET
duration_off_in_ms := _duration_off_in_ms;
END_GET
SET
_duration_off_in_ms := duration_off_in_ms;
END_SET
END_PROPERTY

{attribute 'monitoring' := 'call'}
PROPERTY duration_on : TIME
GET
duration_on := TO_TIME(act_duration_on_in_ms);
END_GET
END_PROPERTY

{attribute 'monitoring' := 'call'}
PROPERTY PUBLIC duration_on_in_ms : ULINT
GET
duration_on_in_ms := _duration_on_in_ms;
END_GET
SET
_duration_on_in_ms := duration_on_in_ms;
END_SET
END_PROPERTY

METHOD PRIVATE init_timestamps
VAR_INPUT
END_VAR
IF timestamp_off_in_ms = 0 AND timestamp_on_in_ms = 0 THEN
  IF signal THEN
    timestamp_on_in_ms := act_timestamp_in_ms;
  ELSE
    timestamp_off_in_ms := act_timestamp_in_ms;
	END_IF
END_IF
END_METHOD

{attribute 'monitoring' := 'call'}
PROPERTY PUBLIC off_is_recording : BOOL
GET
off_is_recording := started_recording AND NOT t_signal_filtertime.Q;
END_GET
END_PROPERTY

{attribute 'monitoring' := 'call'}
PROPERTY off_ratio : REAL
GET
off_ratio := 1.0 - on_ratio;
END_GET
END_PROPERTY

{attribute 'monitoring' := 'call'}
PROPERTY PUBLIC on_is_recording : BOOL
GET
on_is_recording := started_recording AND t_signal_filtertime.Q;
END_GET
END_PROPERTY

{attribute 'monitoring' := 'call'}
PROPERTY on_ratio : REAL
GET
IF (record_duration = T#0S) THEN
  on_ratio := TO_REAL(signal);
ELSE
  on_ratio := TO_REAL(duration_on_in_ms) / TO_REAL(record_duration_in_ms);
END_IF
END_GET
END_PROPERTY

METHOD record
VAR_INPUT
  execute: BOOL;
END_VAR
VAR
  act_timestamp: TIME;
  previous_cycle_time: TIME;
END_VAR
VAR_INST
  previous_timestamp: TIME;
  
  r_signal_filtertime: R_TRIG;
  f_signal: F_TRIG;
  f_execute: F_TRIG;
  r_record_delay: R_TRIG;
END_VAR
f_execute(CLK:=execute);
IF f_execute.Q THEN
  apply_duration();
END_IF
t_record_delay(IN:=execute, PT:=record_delay);

r_record_delay(CLK:=t_record_delay.Q);
IF t_record_delay.Q THEN
  init_timestamps();
  t_signal_filtertime(IN:=signal, PT:=signal_filtertime);
  r_signal_filtertime(CLK:=t_signal_filtertime.Q);
  IF r_signal_filtertime.Q THEN
    apply_duration();
    timestamp_on_in_ms := act_timestamp_in_ms - TO_ULINT(signal_filtertime);
    IF duration_off_in_ms > 0 THEN
      duration_off_in_ms := duration_off_in_ms - TO_ULINT(signal_filtertime);
		END_IF
	END_IF
  f_signal(CLK:=signal);
  IF f_signal.Q OR (r_record_delay.Q AND NOT signal) THEN
    apply_duration();
    timestamp_off_in_ms := act_timestamp_in_ms;
	END_IF
END_IF
END_METHOD

{attribute 'monitoring' := 'call'}
PROPERTY record_delay : TIME
GET
record_delay := _record_delay;
END_GET
SET
_record_delay := record_delay;
END_SET
END_PROPERTY

{attribute 'monitoring' := 'call'}
PROPERTY record_duration : TIME
GET
record_duration := duration_on + duration_off;
END_GET
END_PROPERTY

{attribute 'monitoring' := 'call'}
PROPERTY record_duration_in_ms : ULINT
GET
record_duration_in_ms := duration_on_in_ms + duration_off_in_ms;
END_GET
END_PROPERTY

METHOD reset
VAR_INPUT
END_VAR
duration_off_in_ms := 0;
duration_on_in_ms := 0;
timestamp_off_in_ms := 0;
timestamp_on_in_ms := 0;
END_METHOD

{attribute 'monitoring' := 'call'}
PROPERTY signal : BOOL
GET
signal := _signal;
END_GET
SET
_signal := signal;
END_SET
END_PROPERTY

{attribute 'monitoring' := 'call'}
PROPERTY signal_filtertime : TIME
GET
signal_filtertime := _signal_filtertime;
END_GET
SET
_signal_filtertime := signal_filtertime;
END_SET
END_PROPERTY

{attribute 'monitoring' := 'call'}
PROPERTY started_recording : BOOL
GET
started_recording := t_record_delay.Q;
END_GET
END_PROPERTY

{attribute 'monitoring' := 'call'}
PROPERTY PUBLIC timestamp_off_in_ms : ULINT
GET
timestamp_off_in_ms := _timestamp_off_in_ms;
END_GET
SET
_timestamp_off_in_ms := timestamp_off_in_ms;
END_SET
END_PROPERTY

{attribute 'monitoring' := 'call'}
PROPERTY PUBLIC timestamp_on_in_ms : ULINT
GET
timestamp_on_in_ms := _timestamp_on_in_ms;
END_GET
SET
_timestamp_on_in_ms := timestamp_on_in_ms;
END_SET
END_PROPERTY

END_FUNCTION_BLOCK

// ---- Tests/TestBitAdrState.TcPOU
FUNCTION_BLOCK TestBitAdrState EXTENDS TcUnit.FB_TestSuite
VAR_INPUT
END_VAR
VAR_OUTPUT
END_VAR
VAR
END_VAR

first_bit_of_first_byte_is_off();
first_bit_of_first_byte_is_on();
last_bit_of_first_byte_is_off();
last_bit_of_first_byte_is_on();
first_bit_of_second_byte_is_off();
first_bit_of_second_byte_is_on();
last_bit_of_second_byte_is_off();
last_bit_of_second_byte_is_on();
fourth_bit_of_second_byte_is_on();
out_of_bounds_bit_adr_is_off();

METHOD first_bit_of_first_byte_is_off
VAR
  state: BOOL;
END_VAR
VAR_INST
  b: ARRAY[0..1] OF BYTE;
END_VAR
TEST('first_bit_of_first_byte_is_off');

state := BitAdrState(0, ADR(b), SIZEOF(b));
AssertFalse(state, '');

TEST_FINISHED();
END_METHOD

METHOD first_bit_of_first_byte_is_on
VAR
  state: BOOL;
END_VAR
VAR_INST
  b: ARRAY[0..1] OF BYTE;
END_VAR
TEST('first_bit_of_first_byte_is_on');

b[0] := 1;
state := BitAdrState(0, ADR(b), SIZEOF(b));
AssertTrue(state, '');

TEST_FINISHED();
END_METHOD

METHOD first_bit_of_second_byte_is_off
VAR
  state: BOOL;
END_VAR
VAR_INST
  b: ARRAY[0..1] OF BYTE;
END_VAR
TEST('first_bit_of_second_byte_is_off');

b[1] := 0;
state := BitAdrState(8, ADR(b), SIZEOF(b));
AssertFalse(state, '');

TEST_FINISHED();
END_METHOD

METHOD first_bit_of_second_byte_is_on
VAR
  state: BOOL;
END_VAR
VAR_INST
  b: ARRAY[0..1] OF BYTE;
END_VAR
TEST('first_bit_of_second_byte_is_on');

b[1] := 1;
state := BitAdrState(8, ADR(b), SIZEOF(b));
AssertTrue(state, '');

TEST_FINISHED();
END_METHOD

METHOD fourth_bit_of_second_byte_is_on
VAR
  state: BOOL;
END_VAR
VAR_INST
  b: ARRAY[0..1] OF BYTE;
END_VAR
TEST('fourth_bit_of_second_byte_is_on');

b[1] := 8;
state := BitAdrState(11, ADR(b), SIZEOF(b));
AssertTrue(state, '');

TEST_FINISHED();
END_METHOD

METHOD last_bit_of_first_byte_is_off
VAR
  state: BOOL;
END_VAR
VAR_INST
  b: ARRAY[0..1] OF BYTE;
END_VAR
TEST('last_bit_of_first_byte_is_off');

b[0] := 0;
state := BitAdrState(7, ADR(b), SIZEOF(b));
AssertFalse(state, '');

TEST_FINISHED();
END_METHOD

METHOD last_bit_of_first_byte_is_on
VAR
  state: BOOL;
END_VAR
VAR_INST
  b: ARRAY[0..1] OF BYTE;
END_VAR
TEST('last_bit_of_first_byte_is_on');

b[0] := 128;
state := BitAdrState(7, ADR(b), SIZEOF(b));
AssertTrue(state, '');

TEST_FINISHED();
END_METHOD

METHOD last_bit_of_second_byte_is_off
VAR
  state: BOOL;
END_VAR
VAR_INST
  b: ARRAY[0..1] OF BYTE;
END_VAR
TEST('last_bit_of_second_byte_is_off');

b[1] := 0;
state := BitAdrState(15, ADR(b), SIZEOF(b));
AssertFalse(state, '');

TEST_FINISHED();
END_METHOD

METHOD last_bit_of_second_byte_is_on
VAR
  state: BOOL;
END_VAR
VAR_INST
  b: ARRAY[0..1] OF BYTE;
END_VAR
TEST('last_bit_of_second_byte_is_on');

b[1] := 128;
state := BitAdrState(15, ADR(b), SIZEOF(b));
AssertTrue(state, '');

TEST_FINISHED();
END_METHOD

METHOD out_of_bounds_bit_adr_is_off
VAR
  state: BOOL;
END_VAR
VAR_INST
  b: ARRAY[0..1] OF BYTE;
END_VAR
TEST('out_of_bounds_bit_adr_is_off');

b[0] := 255;
b[1] := 255;
state := BitAdrState(16, ADR(b), SIZEOF(b));
AssertFalse(state, '');

TEST_FINISHED();
END_METHOD

END_FUNCTION_BLOCK

// ---- Object/BitAdrState.TcPOU
FUNCTION BitAdrState : BOOL
VAR_INPUT
  bit_adr: DWORD;
  data_ptr: POINTER TO BYTE;
  data_size: DWORD;
END_VAR
VAR
  index: DINT;
  byte_bit_adr: UDINT;
  byte_mask: BYTE;
END_VAR
VAR CONSTANT
  BYTE_BIT_SIZE: DWORD := 8;
END_VAR

IF bit_adr >= (data_size * BYTE_BIT_SIZE) THEN
  RETURN;
END_IF

index := TRUNC(bit_adr / BYTE_BIT_SIZE);
byte_bit_adr := bit_adr MOD BYTE_BIT_SIZE;
byte_mask := SHL(1, byte_bit_adr);

BitAdrState := (data_ptr[index] AND byte_mask) <> 0;

END_FUNCTION

// ---- Tests/TestModabsInt.TcPOU
FUNCTION_BLOCK TestModabsInt EXTENDS TcUnit.FB_TestSuite
VAR_INPUT
END_VAR
VAR_OUTPUT
END_VAR
VAR
END_VAR

divisor_is_null();
numerator_is_smaller_than_denominator();
numerator_is_negative();
numerator_is_negative_and_bigger_than_denominator();

METHOD divisor_is_null
VAR
  state: INT;
END_VAR
TEST('divisor_is_null');

state := ModabsInt(0, 0);
AssertEquals_INT(0, state, '');

TEST_FINISHED();
END_METHOD

METHOD numerator_is_negative
VAR
  state: INT;
END_VAR
TEST('numerator_is_negative');

state := ModabsInt(-3, 8);
AssertEquals_INT(5, state, '');

TEST_FINISHED();
END_METHOD

METHOD numerator_is_negative_and_bigger_than_denominator
VAR
  state: INT;
END_VAR
TEST('numerator_is_negative_and_bigger_than_denominator');

state := ModabsInt(-9, 8);
AssertEquals_INT(7, state, '');

TEST_FINISHED();
END_METHOD

METHOD numerator_is_smaller_than_denominator
VAR
  state: INT;
END_VAR
TEST('numerator_is_smaller_than_denominator');

state := ModabsInt(4, 8);
AssertEquals_INT(4, state, '');

TEST_FINISHED();
END_METHOD

END_FUNCTION_BLOCK

// ---- Object/ModabsInt.TcPOU
FUNCTION ModabsInt : INT
VAR_INPUT
  val: INT;
  denom: INT;
END_VAR
VAR
  buffer: INT;
END_VAR

IF val < 0 THEN
  val := val + (ABS(val / denom) + 1) * denom;
END_IF
ModabsInt := val MOD denom;

END_FUNCTION

// ---- Timer/GetSystemTimeAsTime.TcPOU
FUNCTION GetSystemTimeAsTime : TIME
VAR_INPUT
END_VAR
VAR
END_VAR

GetSystemTimeAsTime := TO_TIME(F_GetSystemTime() / 10000);

END_FUNCTION

// ---- Timer/SimpleSignalTimeRecorder.TcPOU
FUNCTION_BLOCK SimpleSignalTimeRecorder
VAR_INPUT
END_VAR
VAR_OUTPUT
END_VAR
VAR
  _signal: BOOL;
  
  _duration_in_ms: ULINT;
  _timestamp_in_ms: ULINT;
END_VAR

{attribute 'monitoring' := 'call'}
PROPERTY act_duration_in_ms : ULINT
GET
IF timestamp_in_ms > 0 THEN
  act_duration_in_ms := act_timestamp_in_ms - timestamp_in_ms;
ELSE
  act_duration_in_ms := duration_in_ms;
END_IF
END_GET
END_PROPERTY

{attribute 'monitoring' := 'call'}
PROPERTY PRIVATE act_timestamp_in_ms : ULINT
GET
act_timestamp_in_ms := F_GetSystemTime() / 10000;
END_GET
END_PROPERTY

METHOD PRIVATE apply_duration
VAR_INPUT
END_VAR
IF timestamp_in_ms > 0 THEN
  duration_in_ms := act_duration_in_ms;
  timestamp_in_ms := 0;
END_IF
END_METHOD

{attribute 'monitoring' := 'call'}
PROPERTY duration : TIME
GET
duration := TO_TIME(duration_in_ms);
END_GET
END_PROPERTY

{attribute 'monitoring' := 'call'}
PROPERTY PUBLIC duration_in_ms : ULINT
GET
duration_in_ms := _duration_in_ms;
END_GET
SET
_duration_in_ms := duration_in_ms;
END_SET
END_PROPERTY

METHOD record
VAR_INPUT
  execute: BOOL;
END_VAR
VAR_INST
  r_signal: R_TRIG;
  r_execute: R_TRIG;
  f_execute: F_TRIG;
END_VAR
r_execute(CLK:=execute);
f_execute(CLK:=execute);
IF r_execute.Q AND NOT signal THEN
  timestamp_in_ms := act_timestamp_in_ms;
END_IF
IF f_execute.Q THEN
  timestamp_in_ms := 0;
END_IF

r_signal(CLK:=signal);
IF execute AND r_signal.Q THEN
  apply_duration();
END_IF
END_METHOD

METHOD reset
VAR_INPUT
END_VAR
duration_in_ms := 0;
timestamp_in_ms := 0;
END_METHOD

{attribute 'monitoring' := 'call'}
PROPERTY signal : BOOL
GET
signal := _signal;
END_GET
SET
_signal := signal;
END_SET
END_PROPERTY

{attribute 'monitoring' := 'call'}
PROPERTY PUBLIC timestamp_in_ms : ULINT
GET
timestamp_in_ms := _timestamp_in_ms;
END_GET
SET
_timestamp_in_ms := timestamp_in_ms;
END_SET
END_PROPERTY

END_FUNCTION_BLOCK

// ---- Timer/SimpleTimeRecorder.TcPOU
FUNCTION_BLOCK SimpleTimeRecorder
VAR_INPUT
END_VAR
VAR_OUTPUT
END_VAR
VAR
  _duration_in_ms: ULINT;
  _timestamp_in_ms: ULINT;
END_VAR

{attribute 'monitoring' := 'call'}
PROPERTY act_duration_in_ms : ULINT
GET
IF timestamp_in_ms > 0 THEN
  act_duration_in_ms := act_timestamp_in_ms - timestamp_in_ms;
ELSE
  act_duration_in_ms := duration_in_ms;
END_IF
END_GET
END_PROPERTY

{attribute 'monitoring' := 'call'}
PROPERTY PRIVATE act_timestamp_in_ms : ULINT
GET
act_timestamp_in_ms := F_GetSystemTime() / 10000;
END_GET
END_PROPERTY

METHOD PRIVATE apply_duration
VAR_INPUT
END_VAR
IF timestamp_in_ms > 0 THEN
  duration_in_ms := act_duration_in_ms;
  timestamp_in_ms := 0;
END_IF
END_METHOD

{attribute 'monitoring' := 'call'}
PROPERTY duration : TIME
GET
duration := TO_TIME(duration_in_ms);
END_GET
END_PROPERTY

{attribute 'monitoring' := 'call'}
PROPERTY PUBLIC duration_in_ms : ULINT
GET
duration_in_ms := _duration_in_ms;
END_GET
SET
_duration_in_ms := duration_in_ms;
END_SET
END_PROPERTY

METHOD record
VAR_INPUT
  execute: BOOL;
END_VAR
VAR_INST
  r_signal: R_TRIG;
  r_execute: R_TRIG;
  f_execute: F_TRIG;
END_VAR
r_execute(CLK:=execute);
f_execute(CLK:=execute);
IF r_execute.Q THEN
  timestamp_in_ms := act_timestamp_in_ms;
END_IF
IF f_execute.Q THEN
  apply_duration();
END_IF
END_METHOD

METHOD reset
VAR_INPUT
END_VAR
duration_in_ms := 0;
timestamp_in_ms := 0;
END_METHOD

{attribute 'monitoring' := 'call'}
PROPERTY PUBLIC timestamp_in_ms : ULINT
GET
timestamp_in_ms := _timestamp_in_ms;
END_GET
SET
_timestamp_in_ms := timestamp_in_ms;
END_SET
END_PROPERTY

END_FUNCTION_BLOCK

// ---- Utils/CompareReal.TcPOU
FUNCTION CompareReal : BOOL
VAR_INPUT
  value_1: REAL;
  value_2: REAL;
  tolerance: REAL;
END_VAR
VAR
END_VAR

CompareReal := ABS(value_1 - value_2) <= tolerance;

END_FUNCTION

// ---- Utils/FlashSignal.TcPOU
FUNCTION_BLOCK FlashSignal
VAR_INPUT
  flash_time: TIME;
END_VAR
VAR_OUTPUT
	q: BOOL;
END_VAR
VAR
	timer_flash: TON;
END_VAR

timer_flash(IN:=TRUE, PT:=flash_time);
IF (timer_flash.Q) THEN
	timer_flash(IN:=FALSE);
	q := NOT q;
END_IF

METHOD FB_init : BOOL
VAR_INPUT
	bInitRetains : BOOL; // if TRUE, the retain variables are initialized (warm start / cold start)
	bInCopyCode : BOOL;  // if TRUE, the instance afterwards gets moved into the copy code (online change)
  flash_time: TIME;
END_VAR
THIS^.flash_time := flash_time;
END_METHOD

END_FUNCTION_BLOCK
